// TIA Portal project "GirelloAutomatico" (V15.1)

(* hardware
DEVICE "S7-1200 station_1"  S7-1200 Station
   slot 0: "Telaio di montaggio_0"  S7-1200 Rack  Rack  V1.0
   slot 1: "PLC_1"  CPU 1214C DC/DC/DC  6ES7 214-1AG40-0XB0  V4.2
*)

// ===== PLC "PLC_1"  CPU 1214C DC/DC/DC =====

VAR_GLOBAL   // PLC tag table "Tabella delle variabili standard"
   "P1" AT %I0.1 : Bool;
   "P2" AT %I0.2 : Bool;
   "PG" AT %I0.3 : Bool;
   "PX" AT %I0.4 : Bool;
   "FCS" AT %I0.5 : Bool;
   "FCD" AT %I0.6 : Bool;
   "M1" AT %Q0.0 : Bool;
   "M2" AT %Q0.1 : Bool;
   "MG" AT %Q0.2 : Bool;
   "S" AT %Q0.3 : Bool;
   "D" AT %Q0.4 : Bool;
   "Abilita" AT %I0.0 : Bool;
   "Contatore" AT %MW0 : Int;
END_VAR

DATA_BLOCK "StatoRullo1"   // DB1
{ S7_Optimized_Access := 'TRUE' }
VERSION : 0.1
   VAR RETAIN
      Home : Bool := true;
      RulloScarico : Bool;
      RulloCarico : Bool;
      GirelloScarico : Bool;
      GirelloCarico : Bool;
   END_VAR
BEGIN
END_DATA_BLOCK

DATA_BLOCK "StatoGirello"   // DB2
{ S7_Optimized_Access := 'TRUE' }
VERSION : 0.1
   VAR RETAIN
      Home : Bool := true;
      PosizioneIniziale : Bool;
      GirelloScarico : Bool;
      GirelloCarico : Bool;
      CaricaRullo2 : Bool;
   END_VAR
BEGIN
END_DATA_BLOCK

// folder: System blocks/Program resources

DATA_BLOCK "IEC_Counter_0_DB"   // DB3
{ S7_Optimized_Access := 'TRUE' }
AUTHOR : Simatic
FAMILY : IEC
NAME : CNTR
VERSION : 1.0
// stored: InstanceOfName IEC_COUNTER
"IEC_COUNTER"
BEGIN
END_DATA_BLOCK

// folder: (top level)

ORGANIZATION_BLOCK "Rullo1"   // OB1, LAD, ProgramCycle
TITLE = "Main Program Sweep (Cycle)"
{ S7_Optimized_Access := 'TRUE' }
VERSION : 0.1
   VAR_INPUT
      Initial_Call : Bool;   // Initial call of this OB
      Remanence : Bool;   // =True, if remanent data are available
   END_VAR
BEGIN

REGION Network 1
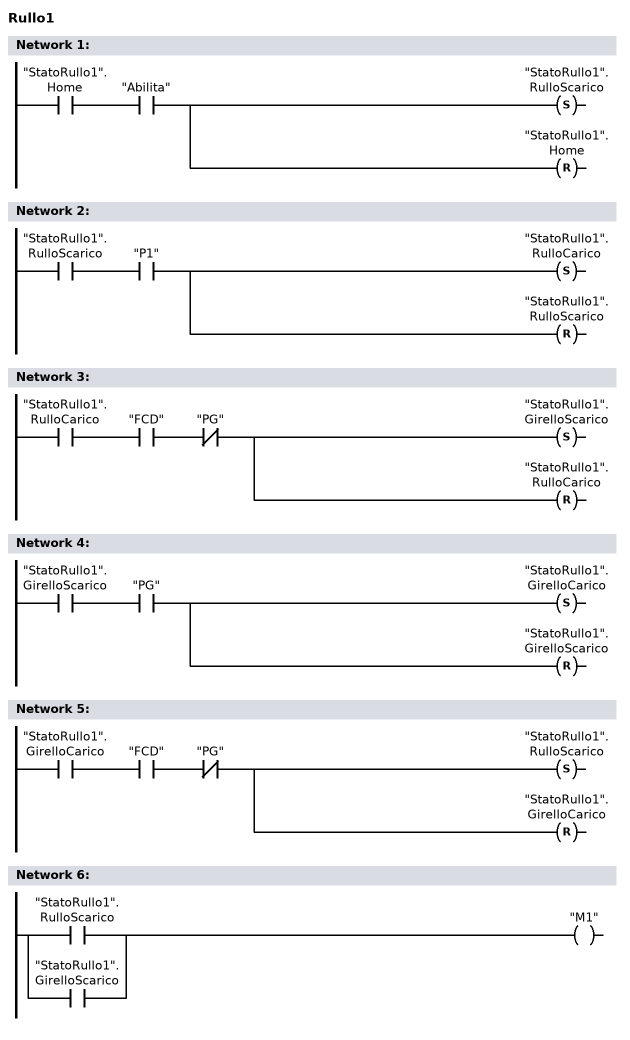
   RUNG wire#powerrail
      Contact( "StatoRullo1".Home )
      Contact( "Abilita" )
      wire#w1
      S_Coil( "StatoRullo1".RulloScarico )
   END_RUNG
   RUNG wire#w1
      R_Coil( "StatoRullo1".Home )
   END_RUNG
   // the same network as SCL:
   IF "StatoRullo1".Home AND "Abilita" THEN
       "StatoRullo1".RulloScarico := TRUE;
       "StatoRullo1".Home := FALSE;
   END_IF;
END_REGION

REGION Network 2
   RUNG wire#powerrail
      Contact( "StatoRullo1".RulloScarico )
      Contact( "P1" )
      wire#w1
      S_Coil( "StatoRullo1".RulloCarico )
   END_RUNG
   RUNG wire#w1
      R_Coil( "StatoRullo1".RulloScarico )
   END_RUNG
   // the same network as SCL:
   IF "StatoRullo1".RulloScarico AND "P1" THEN
       "StatoRullo1".RulloCarico := TRUE;
       "StatoRullo1".RulloScarico := FALSE;
   END_IF;
END_REGION

REGION Network 3
   RUNG wire#powerrail
      Contact( "StatoRullo1".RulloCarico )
      Contact( "FCD" )
      I_Contact( "PG" )
      wire#w1
      S_Coil( "StatoRullo1".GirelloScarico )
   END_RUNG
   RUNG wire#w1
      R_Coil( "StatoRullo1".RulloCarico )
   END_RUNG
   // the same network as SCL:
   IF "StatoRullo1".RulloCarico AND "FCD" AND NOT "PG" THEN
       "StatoRullo1".GirelloScarico := TRUE;
       "StatoRullo1".RulloCarico := FALSE;
   END_IF;
END_REGION

REGION Network 4
   RUNG wire#powerrail
      Contact( "StatoRullo1".GirelloScarico )
      Contact( "PG" )
      wire#w1
      S_Coil( "StatoRullo1".GirelloCarico )
   END_RUNG
   RUNG wire#w1
      R_Coil( "StatoRullo1".GirelloScarico )
   END_RUNG
   // the same network as SCL:
   IF "StatoRullo1".GirelloScarico AND "PG" THEN
       "StatoRullo1".GirelloCarico := TRUE;
       "StatoRullo1".GirelloScarico := FALSE;
   END_IF;
END_REGION

REGION Network 5
   RUNG wire#powerrail
      Contact( "StatoRullo1".GirelloCarico )
      Contact( "FCD" )
      I_Contact( "PG" )
      wire#w1
      S_Coil( "StatoRullo1".RulloScarico )
   END_RUNG
   RUNG wire#w1
      R_Coil( "StatoRullo1".GirelloCarico )
   END_RUNG
   // the same network as SCL:
   IF "StatoRullo1".GirelloCarico AND "FCD" AND NOT "PG" THEN
       "StatoRullo1".RulloScarico := TRUE;
       "StatoRullo1".GirelloCarico := FALSE;
   END_IF;
END_REGION

REGION Network 6
   RUNG wire#powerrail
      Contact( "StatoRullo1".RulloScarico )
      wire#w1
      Coil( "M1" )
   END_RUNG
   RUNG wire#powerrail
      Contact( "StatoRullo1".GirelloScarico )
   END_RUNG wire#w1
   // the same network as SCL:
   "M1" := "StatoRullo1".RulloScarico OR "StatoRullo1".GirelloScarico;
END_REGION
END_ORGANIZATION_BLOCK

ORGANIZATION_BLOCK "Girello"   // OB123, LAD, ProgramCycle
TITLE = "Main Program Sweep (Cycle)"
{ S7_Optimized_Access := 'TRUE' }
VERSION : 0.1
   VAR_INPUT
      Initial_Call : Bool;   // Initial call of this OB
      Remanence : Bool;   // =True, if remanent data are available
   END_VAR
BEGIN

REGION Network 1
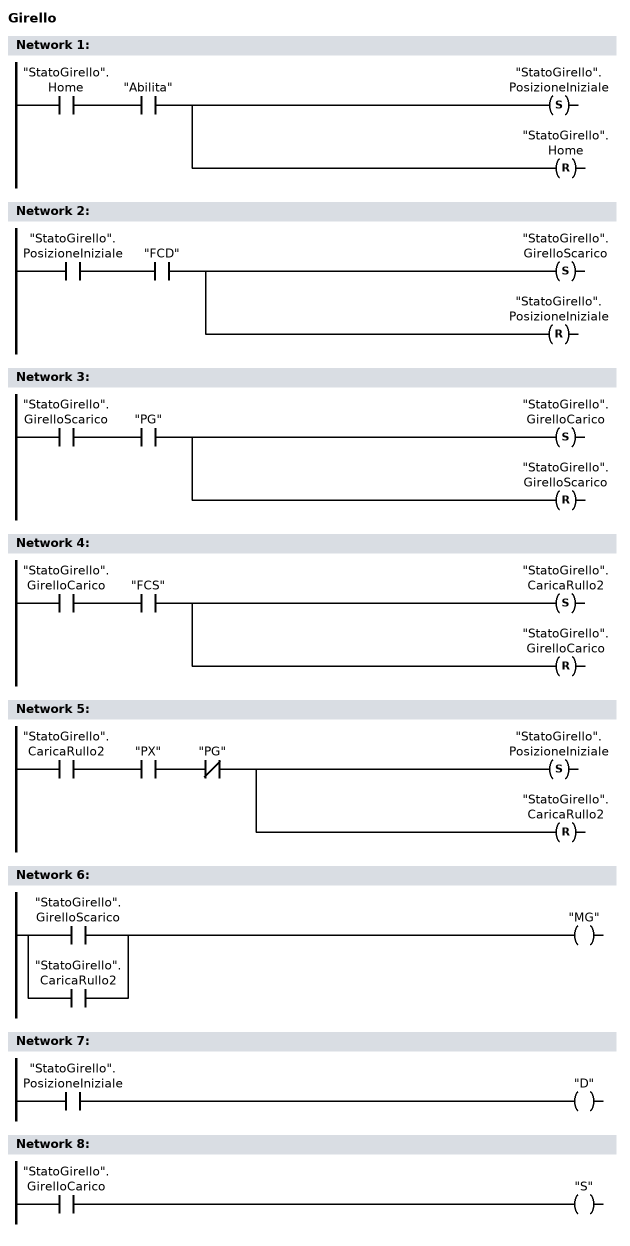
   RUNG wire#powerrail
      Contact( "StatoGirello".Home )
      Contact( "Abilita" )
      wire#w1
      S_Coil( "StatoGirello".PosizioneIniziale )
   END_RUNG
   RUNG wire#w1
      R_Coil( "StatoGirello".Home )
   END_RUNG
   // the same network as SCL:
   IF "StatoGirello".Home AND "Abilita" THEN
       "StatoGirello".PosizioneIniziale := TRUE;
       "StatoGirello".Home := FALSE;
   END_IF;
END_REGION

REGION Network 2
   RUNG wire#powerrail
      Contact( "StatoGirello".PosizioneIniziale )
      Contact( "FCD" )
      wire#w1
      S_Coil( "StatoGirello".GirelloScarico )
   END_RUNG
   RUNG wire#w1
      R_Coil( "StatoGirello".PosizioneIniziale )
   END_RUNG
   // the same network as SCL:
   IF "StatoGirello".PosizioneIniziale AND "FCD" THEN
       "StatoGirello".GirelloScarico := TRUE;
       "StatoGirello".PosizioneIniziale := FALSE;
   END_IF;
END_REGION

REGION Network 3
   RUNG wire#powerrail
      Contact( "StatoGirello".GirelloScarico )
      Contact( "PG" )
      wire#w1
      S_Coil( "StatoGirello".GirelloCarico )
   END_RUNG
   RUNG wire#w1
      R_Coil( "StatoGirello".GirelloScarico )
   END_RUNG
   // the same network as SCL:
   IF "StatoGirello".GirelloScarico AND "PG" THEN
       "StatoGirello".GirelloCarico := TRUE;
       "StatoGirello".GirelloScarico := FALSE;
   END_IF;
END_REGION

REGION Network 4
   RUNG wire#powerrail
      Contact( "StatoGirello".GirelloCarico )
      Contact( "FCS" )
      wire#w1
      S_Coil( "StatoGirello".CaricaRullo2 )
   END_RUNG
   RUNG wire#w1
      R_Coil( "StatoGirello".GirelloCarico )
   END_RUNG
   // the same network as SCL:
   IF "StatoGirello".GirelloCarico AND "FCS" THEN
       "StatoGirello".CaricaRullo2 := TRUE;
       "StatoGirello".GirelloCarico := FALSE;
   END_IF;
END_REGION

REGION Network 5
   RUNG wire#powerrail
      Contact( "StatoGirello".CaricaRullo2 )
      Contact( "PX" )
      I_Contact( "PG" )
      wire#w1
      S_Coil( "StatoGirello".PosizioneIniziale )
   END_RUNG
   RUNG wire#w1
      R_Coil( "StatoGirello".CaricaRullo2 )
   END_RUNG
   // the same network as SCL:
   IF "StatoGirello".CaricaRullo2 AND "PX" AND NOT "PG" THEN
       "StatoGirello".PosizioneIniziale := TRUE;
       "StatoGirello".CaricaRullo2 := FALSE;
   END_IF;
END_REGION

REGION Network 6
   RUNG wire#powerrail
      Contact( "StatoGirello".GirelloScarico )
      wire#w1
      Coil( "MG" )
   END_RUNG
   RUNG wire#powerrail
      Contact( "StatoGirello".CaricaRullo2 )
   END_RUNG wire#w1
   // the same network as SCL:
   "MG" := "StatoGirello".GirelloScarico OR "StatoGirello".CaricaRullo2;
END_REGION

REGION Network 7
   RUNG wire#powerrail
      Contact( "StatoGirello".PosizioneIniziale )
      Coil( "D" )
   END_RUNG
   // the same network as SCL:
   "D" := "StatoGirello".PosizioneIniziale;
END_REGION

REGION Network 8
   RUNG wire#powerrail
      Contact( "StatoGirello".GirelloCarico )
      Coil( "S" )
   END_RUNG
   // the same network as SCL:
   "S" := "StatoGirello".GirelloCarico;
END_REGION
END_ORGANIZATION_BLOCK

ORGANIZATION_BLOCK "Rullo2"   // OB124, LAD, ProgramCycle
TITLE = "Main Program Sweep (Cycle)"
{ S7_Optimized_Access := 'TRUE' }
VERSION : 0.1
   VAR_INPUT
      Initial_Call : Bool;   // Initial call of this OB
      Remanence : Bool;   // =True, if remanent data are available
   END_VAR
BEGIN

REGION Network 1
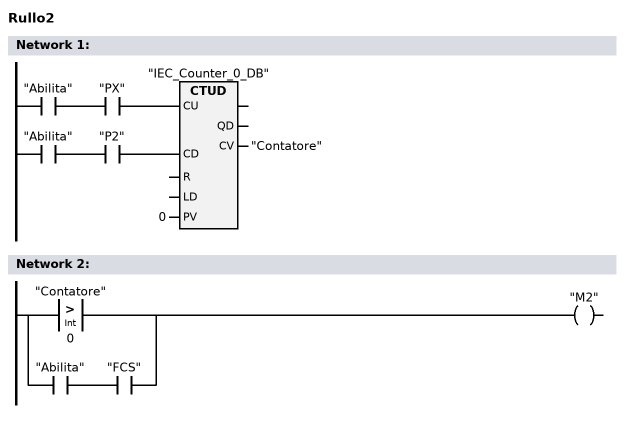
   "IEC_Counter_0_DB".CTUD(CU := "Abilita" AND "PX", CD := "Abilita" AND "P2", PV := 0, CV => "Contatore");
END_REGION

REGION Network 2
   RUNG wire#powerrail
      { S7_Templates := "SrcType := Int" } GT_Contact(in1 := "Contatore", in2 := 0)
      wire#w1
      Coil( "M2" )
   END_RUNG
   RUNG wire#powerrail
      Contact( "Abilita" )
      Contact( "FCS" )
   END_RUNG wire#w1
   // the same network as SCL:
   "M2" := ("Contatore" > 0) OR ("Abilita" AND "FCS");
END_REGION
END_ORGANIZATION_BLOCK